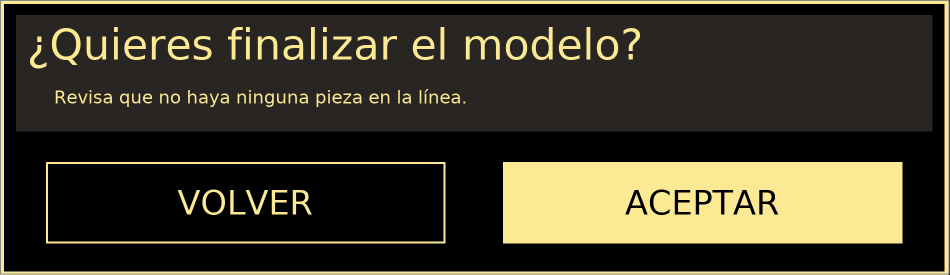
VISUALIZATION V_Emerg_Fin_Prod_Md2  // 950x275
    Rectangle (0,0 948x275)
    Rectangle (16,15 916x116)
    Label (24,17 898x65), "¿Quieres finalizar el modelo?"
    Label (51,85 857x43), "Revisa que no haya ninguna pieza en la línea."
    Rectangle (503,162 399x81), "ACEPTAR", text variable: FuncParoNodoMultidiscos.FunGeneMultidiscos2.P_FinProduccion
        tap FuncParoNodoMultidiscos.FunGeneMultidiscos2.P_FinProduccion
        OnMouseClick: CloseDialog Dialog=V_Emerg_Fin_Prod_Md2, Result=OK, NumpadKeypadSet=True
        OnMouseClick: OpenDialog Dialog=Modelo_Tabla_Md2, OpenModal=True, OpenCentered=True
    Rectangle (46,162 399x81), "VOLVER"
        OnMouseClick: CloseDialog Dialog=V_Emerg_Fin_Prod_Md2, Result=Cancel, NumpadKeypadSet=True
END_VISUALIZATION

(* stored: Version 1.1.0.1, ProductVersion 3.1.4024.12
   Visu V_Emerg_Fin_Prod_Md2: Id {6d75b97d-01f6-4449-b23e-7a4cc7c91ea4} *)
